# EPICS substitutions: kstar/siteApp/TS2/TS2App/Db/ts_mean_B2.substitutions
#
file db/TS_CH_value.db
{
    pattern
        { DEV,    ID,       TAIL,     DESC,                ARG     }

#
        {"B2",    "0",      "MEAN",   "mean value",    "raw_mean"}
        {"B2",    "1",       "MEAN",   "mean value",    "raw_mean"}
        {"B2",    "2",       "MEAN",   "mean value",    "raw_mean"}
        {"B2",    "3",       "MEAN",   "mean value",    "raw_mean"}
        {"B2",    "4",       "MEAN",   "mean value",    "raw_mean"}
        {"B2",    "5",       "MEAN",   "mean value",    "raw_mean"}
        {"B2",    "6",       "MEAN",   "mean value",    "raw_mean"}
        {"B2",    "7",       "MEAN",   "mean value",    "raw_mean"}
        {"B2",    "8",       "MEAN",   "mean value",    "raw_mean"}
        {"B2",    "9",       "MEAN",   "mean value",    "raw_mean"}
        {"B2",    "10",       "MEAN",   "mean value",    "raw_mean"}
        {"B2",    "11",       "MEAN",   "mean value",    "raw_mean"}
        {"B2",    "12",       "MEAN",   "mean value",    "raw_mean"}
        {"B2",    "13",       "MEAN",   "mean value",    "raw_mean"}
        {"B2",    "14",       "MEAN",   "mean value",    "raw_mean"}
        {"B2",    "15",       "MEAN",   "mean value",    "raw_mean"}
#
#
        {"B2",    "0",      "BG_MEAN",   "background mean value",    "bg_mean"}
        {"B2",    "1",      "BG_MEAN",   "background mean value",    "bg_mean"}
        {"B2",    "2",      "BG_MEAN",   "background mean value",    "bg_mean"}
        {"B2",    "3",      "BG_MEAN",   "background mean value",    "bg_mean"}
        {"B2",    "4",      "BG_MEAN",   "background mean value",    "bg_mean"}
        {"B2",    "5",      "BG_MEAN",   "background mean value",    "bg_mean"}
        {"B2",    "6",      "BG_MEAN",   "background mean value",    "bg_mean"}
        {"B2",    "7",      "BG_MEAN",   "background mean value",    "bg_mean"}
        {"B2",    "8",      "BG_MEAN",   "background mean value",    "bg_mean"}
        {"B2",    "9",      "BG_MEAN",   "background mean value",    "bg_mean"}
        {"B2",    "10",      "BG_MEAN",   "background mean value",    "bg_mean"}
        {"B2",    "11",      "BG_MEAN",   "background mean value",    "bg_mean"}
        {"B2",    "12",      "BG_MEAN",   "background mean value",    "bg_mean"}
        {"B2",    "13",      "BG_MEAN",   "background mean value",    "bg_mean"}
        {"B2",    "14",      "BG_MEAN",   "background mean value",    "bg_mean"}
        {"B2",    "15",      "BG_MEAN",   "background mean value",    "bg_mean"}

}
